// TIA Portal V19 export
VAR_GLOBAL   // PLC tag table "D16"
   D16_Lp_EntryReq_LB301 AT %Q200.2 : Bool;   // 256SH1
   D16_Lp_SafetyReset_LB301 AT %Q200.3 : Bool;   // 256SH2
   D16_Pb_EntryReq_LB301 AT %I200.2 : Bool;   // 256SH1
   D16_Pb_SafetyReset_LB301 AT %I200.3 : Bool;   // 256SH2
   D16_Comando_Elettroserratura AT %Q200.0 : Bool;   // 25602
   D16_Funzione_AUX_Elettroserratura AT %Q200.1 : Bool;   // 25605
   D16_Cancello_Chiuso AT %I200.0 : Bool;   // 25601
   D16_Cancello_Bloccato AT %I200.1 : Bool;   // 25603
   D16_Ls_Os1 AT %I1200.1 : Bool;   // 200DI1 - 256A1
   D16_Ls_Os2 AT %I1200.5 : Bool;   // 200DI5 - 256A1
END_VAR
